FUNCTION_BLOCK FB_HMIBase
VAR
	status : ST_HMIStatus;
	configs : ST_HMIConfiguration;
	cmd : ST_HMICommand;
END_VAR

PROPERTY P_Command : ST_HMICommand
GET
P_Command := cmd;
END_GET
SET
cmd := P_Command;
END_SET
END_PROPERTY

PROPERTY P_Configuration : ST_HMIConfiguration
GET
P_Configuration := configs;
END_GET
END_PROPERTY

PROPERTY P_Status : ST_HMIStatus
GET
P_Status := status;
END_GET
SET
status := P_Status;
END_SET
END_PROPERTY

END_FUNCTION_BLOCK

(* stored: Version 1.1.0.1
   POU FB_HMIBase: Id {cccc0bf6-9b64-42bd-b0ca-ff96aa8733e1}, SpecialFunc None
   Property P_Command: Id {38295d4b-cf4d-4043-84fe-a4c04f115626}
   Get Get: Id {9b131594-f8fe-44c4-8bf9-083acf6f22cc}
   Set Set: Id {b2d54d4d-2213-4994-9d02-523a074ae486}
   Property P_Configuration: Id {31ae0e68-4b5e-42f8-9f49-670536860f46}
   Get Get: Id {5871bf39-9c35-4e31-8f00-f8b8922a3e78}
   Property P_Status: Id {f5c47947-7d01-41d6-834a-78421613186a}
   Get Get: Id {10f29e8a-bebe-4e99-ab24-dc1bfc325cde}
   Set Set: Id {a4780232-334c-4510-a907-cfe7552427cb} *)
